PROGRAM timerControl
VAR
	 timer : TOF;  // Timer off-delay function block
END_VAR

// Start the TOF timer if the user moves away (light is still on) and the timer hasn't started
IF GVL.lightStatus = TRUE AND GVL.timerActive = FALSE THEN
    GVL.timerActive := TRUE;
    timer(IN := TRUE, PT := T#15s);  // Start 15-second off-delay timer
END_IF

// If the timer finishes (Q goes TRUE), turn off the light
IF timer.Q THEN
    GVL.lightStatus := FALSE;  // Turn off the light after 15s delay
    GVL.timerActive := FALSE;  // Reset the timer state
END_IF

// Reset the timer when the light is off (if the user moves away before timer completes)
IF GVL.lightStatus = FALSE THEN
    timer(IN := FALSE);  // Stop the timer
    GVL.timerActive := FALSE;  // Reset timer active status
END_IF

END_PROGRAM

(* stored: Version 1.1.0.1, ProductVersion 3.1.4024.12
   POU timerControl: Id {d0c5777f-1fa4-4c4d-ab2e-69154685f57d}, SpecialFunc None *)
